TYPE T_DynamicArrayDataType : ST_Arg; END_TYPE

(* stored: Version 1.1.0.1, ProductVersion 3.1.4024.4
   DUT T_DynamicArrayDataType: Id {25c97d4d-f0e8-4ab0-b7a2-21b45c989e50} *)
